FUNCTION_BLOCK AxisTestSuite
VAR
	StubAxis : AXIS_REF;
	TestAxis : Axis_Base(StubAxis);
 	DummyLogger : Message_Null;
	ObjTestSuite : TestSuite<TestSuiteParameter.MaxTestCount>(ResultFile := JUnitResultFile) := (TestSuiteName := 'Object Test Suite');
END_VAR

AxisPassesEnableRequest_Test();

METHOD AxisPassesEnableRequest_Test
VAR_INST
	Expected : BOOL := TRUE;
	Actual	 : BOOL;
END_VAR
IF ObjTestSuite.Test(__POUNAME()).ExecuteTest() THEN
	Actual := SUCCEEDED(TestAxis.EnableAxis(FALSE,FALSE));
	ObjTestSuite.Test(__POUNAME()).AssertEqual(Expected, Actual);
END_IF
END_METHOD

END_FUNCTION_BLOCK

(* stored: Version 1.1.0.1
   POU AxisTestSuite: Id {0a71268f-cfb2-4598-810c-23a4b39b0a83}, SpecialFunc None
   Method AxisPassesEnableRequest_Test: Id {476e15ea-5203-470c-82e5-b849ce0ce1ae} *)
